// Mitsubishi GX Works2 project: 0.5초 ON , OFF   PLC: Q02/Q02H

PROGRAM MAIN
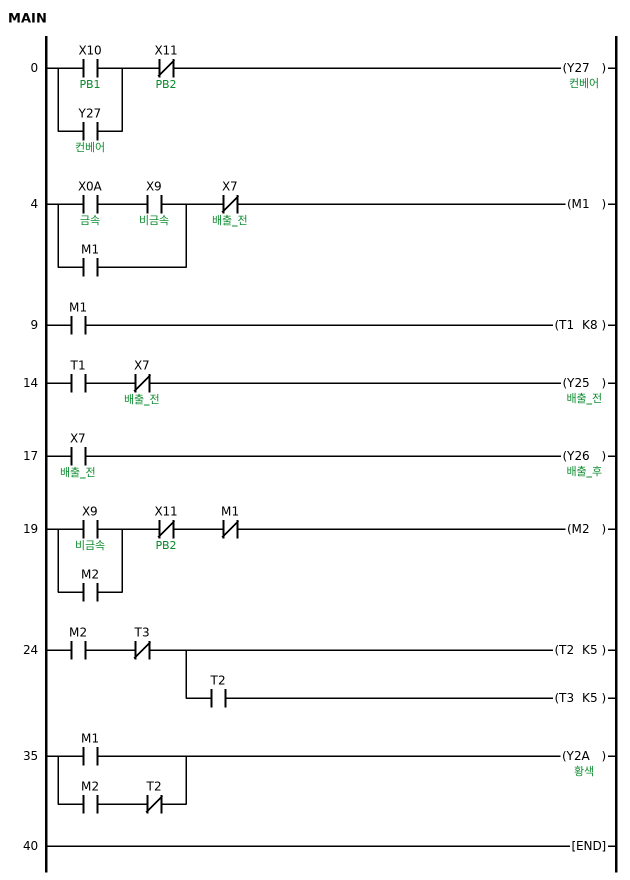
0     LD      X10  ; PB1
      OR      Y27  ; 컨베어
      ANI     X11  ; PB2
      OUT     Y27  ; 컨베어
4     LD      X0A  ; 금속
      AND     X9  ; 비금속
      OR      M1
      ANI     X7  ; 배출_전
      OUT     M1
9     LD      M1
      OUT     T1 K8
14    LD      T1
      ANI     X7  ; 배출_전
      OUT     Y25  ; 배출_전
17    LD      X7  ; 배출_전
      OUT     Y26  ; 배출_후
19    LD      X9  ; 비금속
      OR      M2
      ANI     X11  ; PB2
      ANI     M1
      OUT     M2
24    LD      M2
      ANI     T3
      OUT     T2 K5
      AND     T2
      OUT     T3 K5
35    LD      M1
      LD      M2
      ANI     T2
      ORB
      OUT     Y2A  ; 황색
40    END
END_PROGRAM

// device comments not shown above
X0  ; 공급_후
X1  ; 공급_전
X2  ; 드릴_상
X3  ; 드릴_하
X4  ; 송출_후
X5  ; 송출_전
X6  ; 배출_후
X8  ; 메거진
X12  ; PB3
Y20  ; 공급_전
Y21  ; 공급_후
Y22  ; 드릴_전
Y23  ; 송출_전
Y24  ; 송출_후
Y28  ; 가공드
Y29  ; 적색
Y2B  ; 녹색
